FUNCTION_BLOCK LinearSequence EXTENDS ModuleSequenceBase
VAR_INPUT
	i_primitiveIds: ARRAY [ResiConst.ARR_MIN..ResiConst.MODULE_SEQ_ARR_MAX] OF UINT;
	i_primitiveParams: ARRAY [ResiConst.ARR_MIN..ResiConst.MODULE_SEQ_ARR_MAX] OF ParameterSet;
END_VAR
VAR
	i: UINT;
	
	m_sequenceFinished: BOOL;
	m_primitiveId: UINT;
	m_res: EOperationResult;
END_VAR

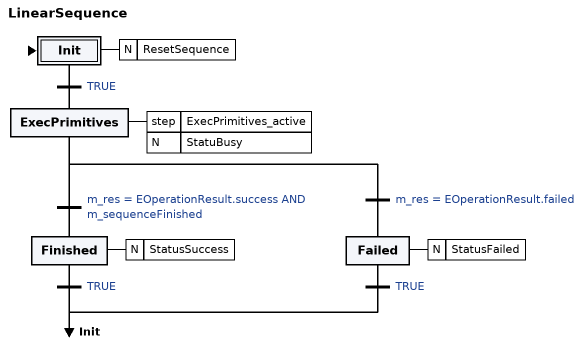
INITIAL_STEP Init:
    ResetSequence(N);
END_STEP
TRANSITION FROM Init TO ExecPrimitives
    := TRUE;
END_TRANSITION
STEP ExecPrimitives:
    ExecPrimitives_active(N);  // step action
    StatuBusy(N);
END_STEP
TRANSITION FROM ExecPrimitives TO Finished
    := m_res = EOperationResult.success AND m_sequenceFinished;
END_TRANSITION
STEP Finished:
    StatusSuccess(N);
END_STEP
TRANSITION FROM Finished TO Init
    := TRUE;
END_TRANSITION
TRANSITION FROM ExecPrimitives TO Failed
    := m_res = EOperationResult.failed;
END_TRANSITION
STEP Failed:
    StatusFailed(N);
END_STEP
TRANSITION FROM Failed TO Init
    := TRUE;
END_TRANSITION

ACTION ExecPrimitives_active:
m_primitiveId := i_primitiveIds[i];

IF m_primitiveId = ESpecialBehaviorIds.empty THEN
	m_sequenceFinished := TRUE;
ELSE
	m_res := m_ptrProcessManager^.Execute(
		i_type := EBehaviorType.control_primitive,
		i_id := m_primitiveId,
		i_params := i_primitiveParams[i]);
		
	IF m_res = EOperationResult.success THEN
		i := i + 1;
	END_IF
END_IF
END_ACTION

PROPERTY Postcondition : IExpression
GET
VAR
	i: UINT;
END_VAR
FOR i := ResiConst.ARR_MIN TO ResiConst.MODULE_SEQ_ARR_MAX DO
	// find the postcondition of the last defined primitive
	IF i_primitiveIds[i] = ESpecialBehaviorIds.empty THEN
		Postcondition := m_ptrProcessManager^.GetBehaviorPtr(EBehaviorType.control_primitive, i_primitiveIds[i - 1])^.Postcondition;
		RETURN;
	END_IF
END_FOR
END_GET
END_PROPERTY

PROPERTY Precondition : IExpression
GET
// precondition of the first defined primitive
Precondition := m_ptrProcessManager^.GetBehaviorPtr(EBehaviorType.control_primitive, i_primitiveIds[ResiConst.ARR_MIN])^.Precondition;
END_GET
END_PROPERTY

METHOD Reset : BOOL
VAR_INPUT
END_VAR
i := ResiConst.ARR_MIN;
m_sequenceFinished := FALSE;
END_METHOD

ACTION ResetSequence:
i := 0;
m_sequenceFinished := FALSE;
m_primitiveId := 0;
o_status := EOperationResult.none;
END_ACTION

ACTION StatuBusy:
o_status := EOperationResult.busy;
END_ACTION

ACTION StatusFailed:
o_status := EOperationResult.failed;
END_ACTION

ACTION StatusSuccess:
o_status := EOperationResult.success;
END_ACTION

END_FUNCTION_BLOCK

(* stored: Version 1.1.0.1, ProductVersion 3.1.4024.12
   POU LinearSequence: Id {8702c906-25d9-45cc-90d7-132d39f8b44d}, SpecialFunc None
   Folder Actions: Id {9966a81d-2c9e-4645-8fd7-65c0464ff9e3}
   Action ExecPrimitives_active: Id {9561d7eb-4465-4dfe-b6d8-ba50f8d8db7c}
   Property Postcondition: Id {8cb0c285-e062-43a5-af68-4fb67e4006f7}
   Get Get: Id {24459118-146b-4609-92eb-c72674a6a854}
   Property Precondition: Id {fc4c39c9-6379-4e6d-9c95-6cf7365fddcc}
   Get Get: Id {cd863e2d-1ce1-4f33-8adc-ce0d53c2c752}
   Method Reset: Id {b4479e0b-fe2c-4250-a7a9-a8eadad6e32b}
   Action ResetSequence: Id {bd1aaad8-f37b-425b-bf42-1b923602b437}
   Action StatuBusy: Id {96f84157-28b4-4154-9ef9-ae2c0a697401}
   Action StatusFailed: Id {4ad365d8-2024-43d2-b7d5-e3d1d976cc37}
   Action StatusSuccess: Id {1293d760-dcda-4b24-a737-a889dc8197cb} *)
